# EPICS substitutions: evrSupport/Db/ioc/IOC-LR20-LS02pattern.substitutions
#
# Pattern records
file evrPatternAll.db {
#	    Device        ,  SLC Pattern Check LNK    , EVR/Trigger
#	                                                  Links
  pattern { DEVICE        ,        LINK4              , LINK5 , LINK6 , TREF }
	  { IOC:LR20:LS02 ,         ""                ,  ""   ,  ""   , 1.03E06 }
}
file evrEventAll.db {
  pattern { DEVICE        }
	  { IOC:LR20:LS02 }
}
